INTERFACE I_State_Object

PROPERTY P_State : eObjectState
GET
END_GET
END_PROPERTY

END_INTERFACE

(* stored: Version 1.1.0.1
   Itf I_State_Object: Id {863ce6eb-0fd9-403d-aa46-80b0f37ebcad}
   Property P_State: Id {9bda4547-8f5e-4062-91ef-9247743ef5b9}
   Get Get: Id {f1871584-17f5-411e-ba06-f74a4c5a52c7} *)
